TYPE ST_ITC_TTQ :
(**************************************************************************************
 * 	Application		:	BoxControl Framework
 *	Revision		:	$Revision: 404529 $
 *	Revision date	:	$Date: 2018-04-23 08:21:38 +0200 (Mo., 23 Apr 2018) $
 *	Last changed by	:	$Author: b7bolm $
 *	URL				:	$URL: http://almscdc.swisslog.com/repo/SWPD/Development/BoxControlFramework/20_Release/trunk/01_Software/BCF/BCF/JumpStart/20_Product/10_App/11_Com/10_Lib/10_Conv/11_ITC/01_DUTs/ST_ITC_TTQ.TcDUT $
 *
 *	Purpose			:	TTQ Structure
 *
 * ------------------------------------------------------------------------------------
 *	Copyright Swisslog [IP AG], Switzerland. All rights reserved.
 * 
 * ------------------------------------------------------------------------------------
 *	
 * 	Revision History: 
 *
 * 	VERSION			DATE			INITIALS			DESCRIPTION
 *	0.1				01.01.2001		swl					Example
 *
 **************************************************************************************)
STRUCT
	Position			: STRING(Conveyor.POSITION_STRINGLENGTH); // 12 Digit SIS Location MM-GGG-EEEE-FF-Z 
	TU_DataIndex		: DINT; // TU-DataIndex
	TU_ID				: STRING(Conveyor.TU_ID_STRINGLENGTH); // 18 Digit SSID
	NbrOfTT				: INT; // Number of TT's
	Label				: STRING(Conveyor.LABEL_LENGTH); // Label length
END_STRUCT
END_TYPE

(* stored: Version 1.1.0.1, ProductVersion 3.1.4022.12
   DUT ST_ITC_TTQ: Id {9d65a934-4ea1-460b-9c6e-785492c11866} *)
